// TIA Portal project "dust_collection" (V15)

(* hardware
DEVICE "S7-1200 station_1"  S7-1200 Station
   slot 0: "Rack_0"  S7-1200 Rack  Rack  V1.0
   slot 1: "PLC_1"  CPU 1214C DC/DC/DC  6ES7 214-1AG40-0XB0  V4.0
DEVICE "HMI_1"  KTP700 Basic PN
   slot 0: "HMI_1"  KTP700 Basic PN  6AV2 123-2GB03-0AX0  15.0.0.0
   slot 1: "HMI_RT_1"  KTP700 Basic PN  6AV2 123-2GB03-0AX0  15.0.0.0
   slot 5: "HMI_1.IE_CP_1"  PROFINET Interface  15.0.0.0
      slot 1: "PROFINET Interface_1"  PROFINET Interface
         slot 1: "Port_1"  Port
*)

// ===== PLC "PLC_1"  CPU 1214C DC/DC/DC =====

VAR_GLOBAL   // PLC tag table "Default tag table"
   "STOP1" AT %I0.0 : Bool;
   "START" AT %I0.1 : Bool;
   "MOTOR1" AT %Q0.0 : Bool;
   "M_KORUMA_1" AT %I1.0 : Bool;
   "STOP2" AT %I0.2 : Bool;
   "START2" AT %I0.3 : Bool;
   "MOTOR2" AT %Q0.1 : Bool;
   "M_KORUMA_2" AT %I1.1 : Bool;
   "STOP3" AT %I0.4 : Bool;
   "START3" AT %I0.5 : Bool;
   "MOTOR3" AT %Q0.2 : Bool;
   "M_KORUMA_3" AT %I1.2 : Bool;
   "STOP4" AT %I0.6 : Bool;
   "START4" AT %I0.7 : Bool;
   "MOTOR4" AT %Q0.3 : Bool;
   "Tag_1" AT %Q0.4 : Bool;
   "M_KORUMA_4" AT %I1.3 : Bool;
   "STOP_01" AT %M0.0 : Bool;
   "START_01" AT %M0.1 : Bool;
   "Stop_02" AT %M0.2 : Bool;
   "Start_02" AT %M0.3 : Bool;
   "Stop_03" AT %M0.4 : Bool;
   "Start_03" AT %M0.5 : Bool;
   "Stop_04" AT %M0.6 : Bool;
   "Start_04" AT %M0.7 : Bool;
END_VAR

ORGANIZATION_BLOCK "Main"   // OB1, LAD, ProgramCycle
TITLE = "Main Program Sweep (Cycle)"
{ S7_Optimized_Access := 'TRUE' }
VERSION : 0.1
// DUST COLLECTION PROJECT
   VAR_INPUT
      Initial_Call : Bool;   // Initial call of this OB
      Remanence : Bool;   // =True, if remanent data are available
   END_VAR
BEGIN

REGION Network 1
   // MOTOR 1 BAŞLATMA DOZOTÖRÜ
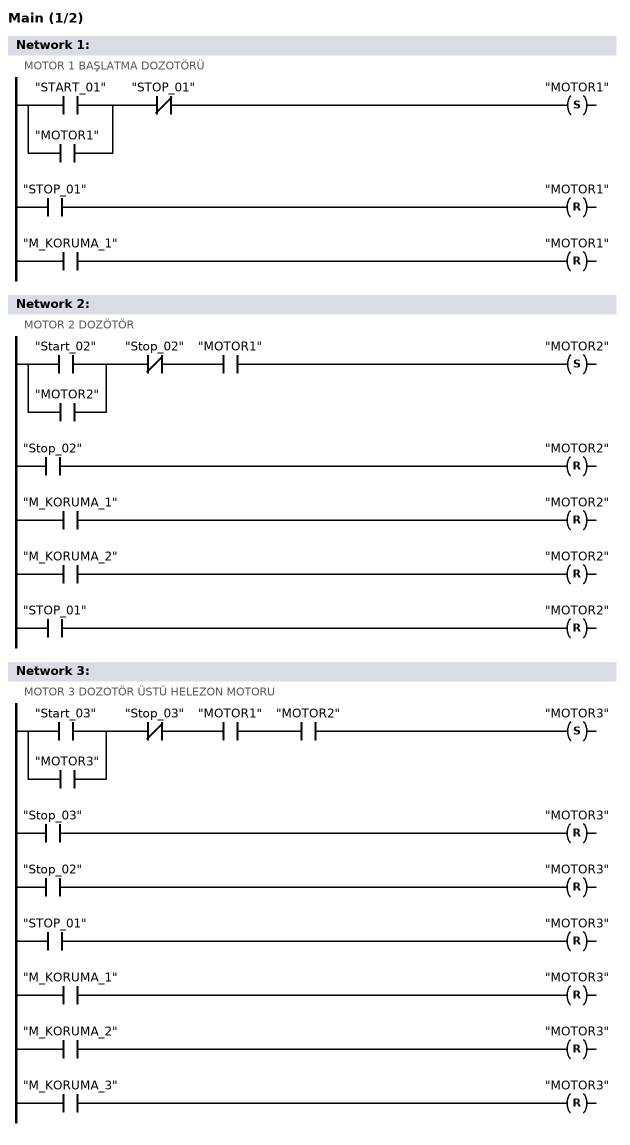
   RUNG wire#powerrail
      Contact( "START_01" )
      wire#w1
      I_Contact( "STOP_01" )
      S_Coil( "MOTOR1" )
   END_RUNG
   RUNG wire#powerrail
      Contact( "MOTOR1" )
   END_RUNG wire#w1
   RUNG wire#powerrail
      Contact( "STOP_01" )
      R_Coil( "MOTOR1" )
   END_RUNG
   RUNG wire#powerrail
      Contact( "M_KORUMA_1" )
      R_Coil( "MOTOR1" )
   END_RUNG
   // the same network as SCL:
   IF ("START_01" OR "MOTOR1") AND NOT "STOP_01" THEN "MOTOR1" := TRUE; END_IF;
   IF "STOP_01" THEN "MOTOR1" := FALSE; END_IF;
   IF "M_KORUMA_1" THEN "MOTOR1" := FALSE; END_IF;
END_REGION

REGION Network 2
   // MOTOR 2 DOZÖTÖR
   RUNG wire#powerrail
      Contact( "Start_02" )
      wire#w1
      I_Contact( "Stop_02" )
      Contact( "MOTOR1" )
      S_Coil( "MOTOR2" )
   END_RUNG
   RUNG wire#powerrail
      Contact( "MOTOR2" )
   END_RUNG wire#w1
   RUNG wire#powerrail
      Contact( "Stop_02" )
      R_Coil( "MOTOR2" )
   END_RUNG
   RUNG wire#powerrail
      Contact( "M_KORUMA_1" )
      R_Coil( "MOTOR2" )
   END_RUNG
   RUNG wire#powerrail
      Contact( "M_KORUMA_2" )
      R_Coil( "MOTOR2" )
   END_RUNG
   RUNG wire#powerrail
      Contact( "STOP_01" )
      R_Coil( "MOTOR2" )
   END_RUNG
   // the same network as SCL:
   IF ("Start_02" OR "MOTOR2") AND NOT "Stop_02" AND "MOTOR1" THEN "MOTOR2" := TRUE; END_IF;
   IF "Stop_02" THEN "MOTOR2" := FALSE; END_IF;
   IF "M_KORUMA_1" THEN "MOTOR2" := FALSE; END_IF;
   IF "M_KORUMA_2" THEN "MOTOR2" := FALSE; END_IF;
   IF "STOP_01" THEN "MOTOR2" := FALSE; END_IF;
END_REGION

REGION Network 3
   // MOTOR 3 DOZOTÖR ÜSTÜ HELEZON MOTORU
   RUNG wire#powerrail
      Contact( "Start_03" )
      wire#w1
      I_Contact( "Stop_03" )
      Contact( "MOTOR1" )
      Contact( "MOTOR2" )
      S_Coil( "MOTOR3" )
   END_RUNG
   RUNG wire#powerrail
      Contact( "MOTOR3" )
   END_RUNG wire#w1
   RUNG wire#powerrail
      Contact( "Stop_03" )
      R_Coil( "MOTOR3" )
   END_RUNG
   RUNG wire#powerrail
      Contact( "Stop_02" )
      R_Coil( "MOTOR3" )
   END_RUNG
   RUNG wire#powerrail
      Contact( "STOP_01" )
      R_Coil( "MOTOR3" )
   END_RUNG
   RUNG wire#powerrail
      Contact( "M_KORUMA_1" )
      R_Coil( "MOTOR3" )
   END_RUNG
   RUNG wire#powerrail
      Contact( "M_KORUMA_2" )
      R_Coil( "MOTOR3" )
   END_RUNG
   RUNG wire#powerrail
      Contact( "M_KORUMA_3" )
      R_Coil( "MOTOR3" )
   END_RUNG
   // the same network as SCL:
   IF ("Start_03" OR "MOTOR3") AND NOT "Stop_03" AND "MOTOR1" AND "MOTOR2" THEN "MOTOR3" := TRUE; END_IF;
   IF "Stop_03" THEN "MOTOR3" := FALSE; END_IF;
   IF "Stop_02" THEN "MOTOR3" := FALSE; END_IF;
   IF "STOP_01" THEN "MOTOR3" := FALSE; END_IF;
   IF "M_KORUMA_1" THEN "MOTOR3" := FALSE; END_IF;
   IF "M_KORUMA_2" THEN "MOTOR3" := FALSE; END_IF;
   IF "M_KORUMA_3" THEN "MOTOR3" := FALSE; END_IF;
END_REGION

REGION Network 4
   // MOTOR 4 132 KW FAN
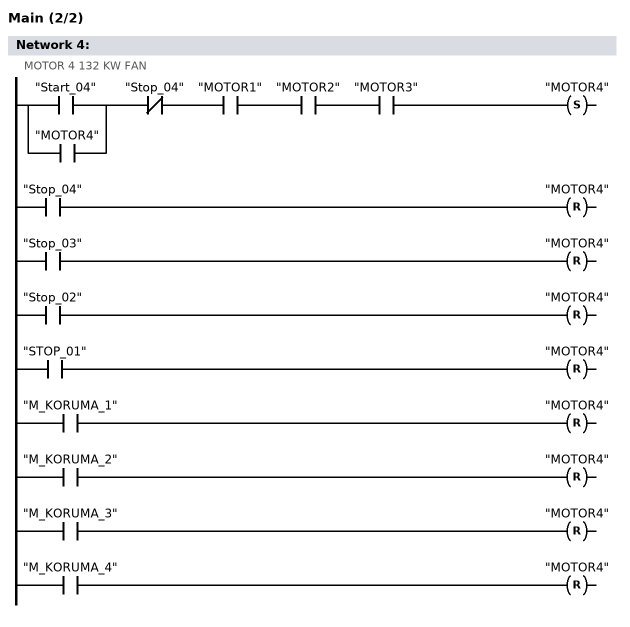
   RUNG wire#powerrail
      Contact( "Start_04" )
      wire#w1
      I_Contact( "Stop_04" )
      Contact( "MOTOR1" )
      Contact( "MOTOR2" )
      Contact( "MOTOR3" )
      S_Coil( "MOTOR4" )
   END_RUNG
   RUNG wire#powerrail
      Contact( "MOTOR4" )
   END_RUNG wire#w1
   RUNG wire#powerrail
      Contact( "Stop_04" )
      R_Coil( "MOTOR4" )
   END_RUNG
   RUNG wire#powerrail
      Contact( "Stop_03" )
      R_Coil( "MOTOR4" )
   END_RUNG
   RUNG wire#powerrail
      Contact( "Stop_02" )
      R_Coil( "MOTOR4" )
   END_RUNG
   RUNG wire#powerrail
      Contact( "STOP_01" )
      R_Coil( "MOTOR4" )
   END_RUNG
   RUNG wire#powerrail
      Contact( "M_KORUMA_1" )
      R_Coil( "MOTOR4" )
   END_RUNG
   RUNG wire#powerrail
      Contact( "M_KORUMA_2" )
      R_Coil( "MOTOR4" )
   END_RUNG
   RUNG wire#powerrail
      Contact( "M_KORUMA_3" )
      R_Coil( "MOTOR4" )
   END_RUNG
   RUNG wire#powerrail
      Contact( "M_KORUMA_4" )
      R_Coil( "MOTOR4" )
   END_RUNG
   // the same network as SCL:
   IF ("Start_04" OR "MOTOR4") AND NOT "Stop_04" AND "MOTOR1" AND "MOTOR2" AND "MOTOR3" THEN
       "MOTOR4" := TRUE;
   END_IF;
   IF "Stop_04" THEN "MOTOR4" := FALSE; END_IF;
   IF "Stop_03" THEN "MOTOR4" := FALSE; END_IF;
   IF "Stop_02" THEN "MOTOR4" := FALSE; END_IF;
   IF "STOP_01" THEN "MOTOR4" := FALSE; END_IF;
   IF "M_KORUMA_1" THEN "MOTOR4" := FALSE; END_IF;
   IF "M_KORUMA_2" THEN "MOTOR4" := FALSE; END_IF;
   IF "M_KORUMA_3" THEN "MOTOR4" := FALSE; END_IF;
   IF "M_KORUMA_4" THEN "MOTOR4" := FALSE; END_IF;
END_REGION
END_ORGANIZATION_BLOCK

(* ===== HMI "HMI_RT_1" =====
system functions are stored by id; their names below are inferred from use
connection "HMI_Connection_1": ETHERNET, SMART_S7_1200_OMS

HMI tags "Default tag table"
   "Tag_ScreenNumber" : UInt, internal
   "START" : Bool = PLC START AT %I0.1, 1 s
   "STOP1" : Bool = PLC STOP1 AT %I0.0, 1 s
   "START2" : Bool = PLC START2 AT %I0.3, 1 s
   "STOP2" : Bool = PLC STOP2 AT %I0.2, 1 s
   "START3" : Bool = PLC START3 AT %I0.5, 1 s
   "STOP3" : Bool = PLC STOP3 AT %I0.4, 1 s
   "START4" : Bool = PLC START4 AT %I0.7, 1 s
   "STOP4" : Bool = PLC STOP4 AT %I0.6, 1 s
   "MOTOR1" : Bool = PLC MOTOR1 AT %Q0.0, 1 s
   "MOTOR2" : Bool = PLC MOTOR2 AT %Q0.1, 1 s
   "MOTOR3" : Bool = PLC MOTOR3 AT %Q0.2, 1 s
   "MOTOR4" : Bool = PLC MOTOR4 AT %Q0.3, 1 s
   "START_01" : Bool = PLC START_01 AT %M0.1, 1 s
   "STOP_01" : Bool = PLC STOP_01 AT %M0.0, 1 s
   "Start_02" : Bool = PLC Start_02 AT %M0.3, 1 s
   "Stop_02" : Bool = PLC Stop_02 AT %M0.2, 1 s
   "Start_03" : Bool = PLC Start_03 AT %M0.5, 1 s
   "Stop_03" : Bool = PLC Stop_03 AT %M0.4, 1 s
   "Start_04" : Bool = PLC Start_04 AT %M0.7, 1 s
   "Stop_04" : Bool = PLC Stop_04 AT %M0.6, 1 s

Template "Template_1" 800x480
   Button "Exit" at 714,429 size 71x50; TextOff 'Exit'; PictureOff "ExitRuntime_KTP700_Basic_PN_TR"; PictureOn "ExitRuntime_KTP700_Basic_PN_TR"
      on Release: StopRuntime(0)
   Button "Template_Button" at 614,429 size 71x50; TextOff 'Text'
   Button "Template_Button_1" at 514,429 size 71x50; TextOff 'Text'
   Button "Template_Button_2" at 414,429 size 71x50; TextOff 'Text'
   Button "Template_Button_3" at 314,429 size 71x50; TextOff 'Text'
   Button "Template_Button_4" at 214,429 size 71x50; TextOff 'Text'
   Button "Template_Button_5" at 114,429 size 71x50; TextOff 'Text'
   Button "Start screen" at 14,429 size 71x50; TextOff 'Start screen'; PictureOff "NavigateHome_KTP700_Basic_PN_TR"; PictureOn "NavigateHome_KTP700_Basic_PN_TR"
      on Release: ActivateScreen("Root screen", 0)
   SymbolicIOField "Symbolic_IO_Field_Screen" at 2,9 size 691x33; TextOff '0'; TextOn '1'; TextList "TextList_ScreenNames"
      ProcessValue <- "Tag_ScreenNumber"
      on Change: ActivateScreenByNumber("Tag_ScreenNumber", 0)
   DateTimeField "HmiScreenItemData" at 695,25 size 105x25
   DateTimeField "HmiScreenItemData_1" at 695,0 size 105x25

screen "Root screen" 800x480, template "Template_1"
   on GenerateScreen: SetTag("Tag_ScreenNumber", 1)
   Button "Button_1" at 44,98 size 96x32; TextOff 'START'
      on Press: SetBit("START_01")
      on Release: ResetBit("START_01")
   Button "Button_2" at 173,98 size 96x32; TextOff 'STOP'
      on Press: SetBit("STOP_01")
      on Release: ResetBit("STOP_01")
   Button "Button_3" at 486,97 size 96x32; TextOff 'START'
      on Press: SetBit("Start_02")
      on Release: ResetBit("Start_02")
   Button "Button_4" at 626,98 size 96x32; TextOff 'STOP'
      on Press: SetBit("Stop_02")
      on Release: ResetBit("Stop_02")
   Button "Button_5" at 44,282 size 96x32; TextOff 'START'
      on Release: ResetBit("Start_03")
      on Press: SetBit("Start_03")
   Button "Button_6" at 177,282 size 96x32; TextOff 'STOP'
      on Press: SetBit("Stop_03")
      on Release: ResetBit("Stop_03")
   Button "Button_7" at 488,278 size 96x32; TextOff 'START'
      on Press: SetBit("Start_04")
      on Release: ResetBit("Start_04")
   Button "Button_8" at 632,278 size 96x32; TextOff 'STOP'
      on Press: SetBit("Stop_04")
      on Release: ResetBit("Stop_04")
   TextField "Text field_1" at 37,62 size 275x23; Text 'MOTOR 1 BAŞLATMA DOZOTÖRÜ'
   TextField "Text field_2" at 534,59 size 167x23; Text 'MOTOR 2 DOZOTÖR'
   TextField "Text field_3" at 17,236 size 370x23; Text 'MOTOR3 DOZOTÖR ÜSTÜ HELEZON MOTORU'
   TextField "Text field_4" at 516,238 size 186x23; Text 'MOTOR 4 132 KW FAN'
   Circle "Circle_2" at 583,152 size 48x48
      Appearance <- "MOTOR2"
   Circle "Circle_3" at 126,338 size 48x48
      Appearance <- "MOTOR3"
   Circle "Circle_4" at 582,338 size 48x48
      Appearance <- "MOTOR4"
   Circle "Circle_1" at 124,160 size 48x48
      Appearance <- "MOTOR1"
*)